// TwinCAT 3 PLC project vision
// ProgramVersion: 3.1.4023.0
// libraries:
//   Tc2_Standard, * (Beckhoff Automation GmbH)
//   Tc2_System, * (Beckhoff Automation GmbH)
//   Tc3_Module, * (Beckhoff Automation GmbH)
//   Tc3_Vision, * (Beckhoff Automation GmbH)
// project tree:
//   / PlcTask.TcTTO
//   POUs/ MAIN.TcPOU
// real-time tasks:
//   TASK PlcTask: cycle T#10ms, priority 20, ADS port 350
//   TASK VnTask ImgAcq (Camera1): cycle T#1ms, priority 5, ADS port 351
//   TASK VnTask ADS (Camera1): cycle T#10ms, priority 6, ADS port 352
//   TASK VnTask ImgAcq (Camera1-1): cycle T#1ms, priority 7, ADS port 353
//   TASK VnTask ADS (Camera1-1): cycle T#10ms, priority 8, ADS port 354
//   TASK VnTask ImgAcq (Camera1-2): cycle T#1ms, priority 9, ADS port 355
//   TASK VnTask ADS (Camera1-2): cycle T#10ms, priority 10, ADS port 356
//   TASK VnTask ImgAcq (Camera2): cycle T#1ms, priority 12, ADS port 357
//   TASK VnTask ADS (Camera2): cycle T#10ms, priority 13, ADS port 358
// I/O:
//   DEVICE Device 1 (RT-Ethernet Adapter)

CONFIGURATION vision
    RESOURCE PLC ON TwinCAT3
        TASK PlcTask(INTERVAL := T#10ms, PRIORITY := 20);
    END_RESOURCE
END_CONFIGURATION

// ---- POUs/MAIN.TcPOU
PROGRAM MAIN
VAR
	hr: HRESULT;
	fbCamera: FB_VN_SimpleCameraControl;
	eState: ETcVnCameraState;
	
	ipImageIn: ITcVnImage;
	ipImageInDisp: ITcVnDisplayableImage;
END_VAR

eState:= fbCamera.GetState();

CASE eState OF 
	TCVN_CS_INITIAL, TCVN_CS_OPENING, TCVN_CS_OPENED, TCVN_CS_STARTACQUISITION:
	hr:=fbCamera.StartAcquisition();
	
	TCVN_CS_ACQUIRING:
	hr:= fbCamera.GetCurrentImage(ipImageIn);
	hr:= F_VN_CopyIntoDisplayableImage(ipImageIn, ipImageInDisp, hr);
	
	TCVN_CS_ERROR:
	hr:= fbCamera.Reset();
	
	
END_CASE

END_PROGRAM
